// TIA Portal V17 export
// export: Created 2026-04-13T11:12:44.7392036Z, ExportSetting WithDefaults, DisplayName Totally Integrated Automation Portal, DisplayVersion V17 Update 4, DisplayName TIA Portal Openness, DisplayVersion V17 Update 4, DisplayName TIA Portal Version Control Interface, DisplayVersion V17, DisplayName SINAMICS Startdrive Advanced, DisplayVersion V17, DisplayName SINAMICS Startdrive G130, G150, S120, S150, SINAMICS MV, S210, DisplayVersion V17, DisplayName SINAMICS Startdrive G110M, G120, G120C, G120D, G120P, G115D, DisplayVersion V17, DisplayName STEP 7 Professional, DisplayVersion V17 Update 4, DisplayName STEP 7 Safety, DisplayVersion V17, DisplayName WinCC Professional, DisplayVersion V17 Update 4
DATA_BLOCK "OUTCIPZS"   // DB47
{ S7_Optimized_Access := 'TRUE' }
VERSION : 0.1
// stored: AutoNumber true, DBAccessibleFromOPCUA true, DBAccessibleFromWebserver true, IsOnlyStoredInLoadMemory false, IsRetainMemResEnabled false, IsWriteProtectedInAS false, MemoryReserve 100
   VAR RETAIN
      "1设定时间" : Real := 10.0;
      "2设定时间" : Real := 10.0;
      "3设定时间" : Real := 10.0;
      "4设定时间" : Real := 10.0;
      "5设定时间" : Real := 10.0;
      "6设定时间" : Real := 10.0;
      "7设定时间" : Real := 10.0;
      "8设定时间" : Real := 10.0;
      "9设定时间" : Real := 10.0;
      "10设定时间" : Real := 10.0;
      "11设定时间" : Real := 10.0;
      "12设定时间" : Real := 10.0;
      "13设定时间" : Real := 10.0;
      "14设定时间" : Real := 10.0;
      "15设定时间" : Real := 10.0;
      "16设定时间" : Real := 10.0;
   END_VAR
   VAR
      "1计时" : Real;
      "2计时" : Real;
      "3计时" : Real;
      "4计时" : Real;
      "5计时" : Real;
      "6计时" : Real;
      "7计时" : Real;
      "8计时" : Real;
      "9计时" : Real;
      "10计时" : Real;
      "11计时" : Real;
      "12计时" : Real;
      "13计时" : Real;
      "14计时" : Real;
      "15计时" : Real;
      "16计时" : Real;
   END_VAR
BEGIN
END_DATA_BLOCK
